TYPE ST_GC_CtrlStatus :
STRUCT
	ModuleCtrl : ST_ModuleCtrl;
	ServiceCtrl : ST_GC_ServiceCtrl;
	ECID : ST_GC_ECID;
	
	ModuleStatus : ST_ModuleStatus;
	ServiceStatus : ST_GC_ServiceStatus;
	SVID : ST_GC_SVID;
END_STRUCT
END_TYPE

(* stored: Version 1.1.0.1, ProductVersion 3.1.4026.18
   DUT ST_GC_CtrlStatus: Id {5bc49452-96f1-4f35-9aa8-ce0a3acfe375} *)
